{attribute 'qualified_only'}
{attribute 'strict'}
{attribute 'to_string'}
TYPE E_MCS2HomeMethod :
(
    AutoMethod := -1,
    CurrentPositionMethod := 37
)SINT;
END_TYPE

(* stored: Version 1.1.0.1
   DUT E_MCS2HomeMethod: Id {41f01279-2525-481d-bbe4-4e1ce0c8d9ff} *)
